TYPE E_DayPLShort :(Pn:=1, Wt, SR, Cz, Pt, So, N);
END_TYPE

(* stored: Version 1.1.0.1, ProductVersion 3.1.4019.2
   DUT E_DayPLShort: Id {d4825304-34eb-47d6-a6d1-415586ed0281} *)
